TYPE TelemetryRelativeHumiditiesConfig :
STRUCT
	///Relative humidity of the air at the top of the tube
	topAir: MeasurementConfig;
	///Relative humidity of the air inside the tube
	insideTube: MeasurementConfig;
END_STRUCT
END_TYPE

(* stored: Version 1.1.0.1, ProductVersion 3.1.4019.2
   DUT TelemetryRelativeHumiditiesConfig: Id {c8055a4f-7c80-4d80-bfe2-e01eb88fad4a} *)
